ABB RAPID module: P700.mod

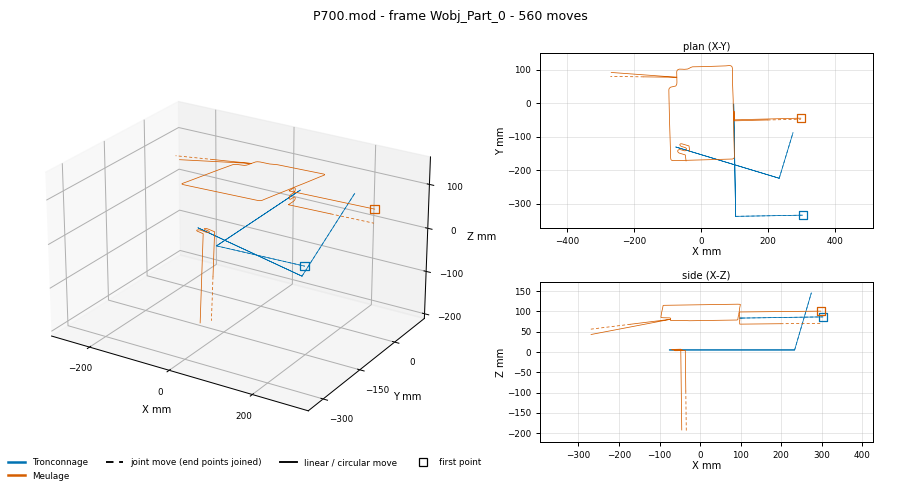
[picture p0: tool path of P700.mod in frame Wobj_Part_0, 560 of 580 moves have a stored position in this frame; points joined in program order, loops and branches not executed]
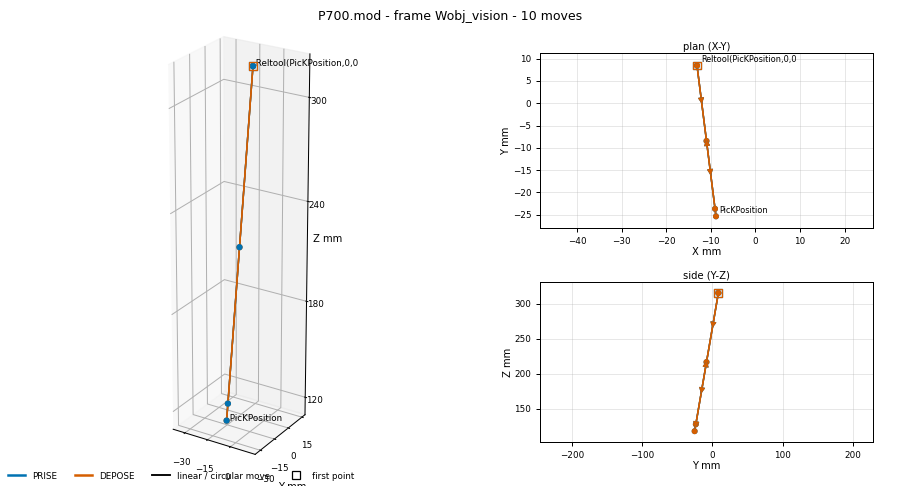
[picture p1: tool path of P700.mod in frame Wobj_vision, 10 of 580 moves have a stored position in this frame; points joined in program order, loops and branches not executed]
MODULE P700

    ! Nom         :P700
    ! Description :
    ! Créé le     :25/05/2023 15:43:03

    LOCAL CONST SPEEDDATA VitesseLente :=[10,500,0,0];
	LOCAL CONST SPEEDDATA VitesseRapide :=[30,500,0,0];
    !
    !Point de prise
    LOCAL PERS Robtarget PicKPosition := [[-8.82508252387174,-25.3604608008818,118.073527161625],[0.0672015502664613,0.699628699637396,0.709367418327075,-0.0529291989496386],[0,0,0,0],[8.999999E+09,8.999999E+09,8.999999E+09,8.999999E+09,8.999999E+09,8.999999E+09]];
	LOCAL PERS Pose Ref := [[0,0,0],[1,0,0,0]];
    !
    !Declaration des points de meulage

    !Tr_meulage_motif_1 : Meulage d'un motif
    LOCAL CONST Robtarget Tr_meulage_motif_1_0 := [[97.6019453125,-49.17523046875,98.798203125],[0.491182031399638,-0.496295254779522,-0.508791654884103,0.50354968377882],[0,0,0,0],[8.999999E+09,8.999999E+09,8.999999E+09,8.999999E+09,8.999999E+09,8.999999E+09]];
    LOCAL CONST Robtarget Tr_meulage_motif_1_1 := [[97.584328125,-48.1753828125,98.7986484375],[0.491182031399638,-0.496295254779522,-0.508791654884103,0.50354968377882],[0,0,0,0],[8.999999E+09,8.999999E+09,8.999999E+09,8.999999E+09,8.999999E+09,8.999999E+09]];
    LOCAL CONST Robtarget Tr_meulage_motif_1_2 := [[97.56671875,-47.1755390625,98.7991015625],[0.491182031399638,-0.496295254779522,-0.508791654884103,0.50354968377882],[0,0,0,0],[8.999999E+09,8.999999E+09,8.999999E+09,8.999999E+09,8.999999E+09,8.999999E+09]];
    LOCAL CONST Robtarget Tr_meulage_motif_1_3 := [[97.549109375,-46.1756953125,98.7995546875],[0.491182031399638,-0.496295254779522,-0.508791654884103,0.50354968377882],[0,0,0,0],[8.999999E+09,8.999999E+09,8.999999E+09,8.999999E+09,8.999999E+09,8.999999E+09]];
    LOCAL CONST Robtarget Tr_meulage_motif_1_4 := [[97.5314921875,-45.1758515625,98.8],[0.491182031399638,-0.496295254779522,-0.508791654884103,0.50354968377882],[0,0,0,0],[8.999999E+09,8.999999E+09,8.999999E+09,8.999999E+09,8.999999E+09,8.999999E+09]];
    LOCAL CONST Robtarget Tr_meulage_motif_1_5 := [[97.5138828125,-44.17600390625,98.800453125],[0.491182031399638,-0.496295254779522,-0.508791654884103,0.50354968377882],[0,0,0,0],[8.999999E+09,8.999999E+09,8.999999E+09,8.999999E+09,8.999999E+09,8.999999E+09]];
    LOCAL CONST Robtarget Tr_meulage_motif_1_6 := [[97.4962734375,-43.17616015625,98.80090625],[0.491182031399638,-0.496295254779522,-0.508791654884103,0.50354968377882],[0,0,0,0],[8.999999E+09,8.999999E+09,8.999999E+09,8.999999E+09,8.999999E+09,8.999999E+09]];
    LOCAL CONST Robtarget Tr_meulage_motif_1_7 := [[97.47865625,-42.17631640625,98.801359375],[0.491182031399638,-0.496295254779522,-0.508791654884103,0.50354968377882],[0,0,0,0],[8.999999E+09,8.999999E+09,8.999999E+09,8.999999E+09,8.999999E+09,8.999999E+09]];
    LOCAL CONST Robtarget Tr_meulage_motif_1_8 := [[97.461046875,-41.17647265625,98.8018046875],[0.491182031399638,-0.496295254779522,-0.508791654884103,0.50354968377882],[0,0,0,0],[8.999999E+09,8.999999E+09,8.999999E+09,8.999999E+09,8.999999E+09,8.999999E+09]];
    LOCAL CONST Robtarget Tr_meulage_motif_1_9 := [[97.4434296875,-40.176625,98.8022578125],[0.491182031399638,-0.496295254779522,-0.508791654884103,0.50354968377882],[0,0,0,0],[8.999999E+09,8.999999E+09,8.999999E+09,8.999999E+09,8.999999E+09,8.999999E+09]];
    LOCAL CONST Robtarget Tr_meulage_motif_1_10 := [[97.4258203125,-39.17678125,98.8027109375],[0.491182031399638,-0.496295254779522,-0.508791654884103,0.50354968377882],[0,0,0,0],[8.999999E+09,8.999999E+09,8.999999E+09,8.999999E+09,8.999999E+09,8.999999E+09]];
    LOCAL CONST Robtarget Tr_meulage_motif_1_11 := [[97.4082109375,-38.1769375,98.80315625],[0.491182031399638,-0.496295254779522,-0.508791654884103,0.50354968377882],[0,0,0,0],[8.999999E+09,8.999999E+09,8.999999E+09,8.999999E+09,8.999999E+09,8.999999E+09]];
    LOCAL CONST Robtarget Tr_meulage_motif_1_12 := [[97.39059375,-37.17709375,98.803609375],[0.491182031399638,-0.496295254779522,-0.508791654884103,0.50354968377882],[0,0,0,0],[8.999999E+09,8.999999E+09,8.999999E+09,8.999999E+09,8.999999E+09,8.999999E+09]];
    LOCAL CONST Robtarget Tr_meulage_motif_1_13 := [[97.372984375,-36.17724609375,98.8040625],[0.491182031399638,-0.496295254779522,-0.508791654884103,0.50354968377882],[0,0,0,0],[8.999999E+09,8.999999E+09,8.999999E+09,8.999999E+09,8.999999E+09,8.999999E+09]];
    LOCAL CONST Robtarget Tr_meulage_motif_1_14 := [[97.3553671875,-35.17740234375,98.8045078125],[0.491182031399638,-0.496295254779522,-0.508791654884103,0.50354968377882],[0,0,0,0],[8.999999E+09,8.999999E+09,8.999999E+09,8.999999E+09,8.999999E+09,8.999999E+09]];
    LOCAL CONST Robtarget Tr_meulage_motif_1_15 := [[97.3377578125,-34.17755859375,98.8049609375],[0.491182031399638,-0.496295254779522,-0.508791654884103,0.50354968377882],[0,0,0,0],[8.999999E+09,8.999999E+09,8.999999E+09,8.999999E+09,8.999999E+09,8.999999E+09]];
    LOCAL CONST Robtarget Tr_meulage_motif_1_16 := [[97.3201484375,-33.1777109375,98.8054140625],[0.491182031399638,-0.496295254779522,-0.508791654884103,0.50354968377882],[0,0,0,0],[8.999999E+09,8.999999E+09,8.999999E+09,8.999999E+09,8.999999E+09,8.999999E+09]];
    LOCAL CONST Robtarget Tr_meulage_motif_1_17 := [[97.30253125,-32.1778671875,98.805859375],[0.491182031399638,-0.496295254779522,-0.508791654884103,0.50354968377882],[0,0,0,0],[8.999999E+09,8.999999E+09,8.999999E+09,8.999999E+09,8.999999E+09,8.999999E+09]];
    LOCAL CONST Robtarget Tr_meulage_motif_1_18 := [[97.284921875,-31.1780234375,98.8063125],[0.491182031399638,-0.496295254779522,-0.508791654884103,0.50354968377882],[0,0,0,0],[8.999999E+09,8.999999E+09,8.999999E+09,8.999999E+09,8.999999E+09,8.999999E+09]];
    LOCAL CONST Robtarget Tr_meulage_motif_1_19 := [[97.2673046875,-30.178177734375,98.806765625],[0.491182031399638,-0.496295254779522,-0.508791654884103,0.50354968377882],[0,0,0,0],[8.999999E+09,8.999999E+09,8.999999E+09,8.999999E+09,8.999999E+09,8.999999E+09]];
    LOCAL CONST Robtarget Tr_meulage_motif_1_20 := [[97.2514296875,-29.18569140625,98.6966328125],[0.491182031399638,-0.496295254779522,-0.508791654884103,0.50354968377882],[0,0,0,0],[8.999999E+09,8.999999E+09,8.999999E+09,8.999999E+09,8.999999E+09,8.999999E+09]];
    LOCAL CONST Robtarget Tr_meulage_motif_1_21 := [[97.237828125,-28.239189453125,98.485890625],[0.491182031399638,-0.496295254779522,-0.508791654884103,0.50354968377882],[0,0,0,0],[8.999999E+09,8.999999E+09,8.999999E+09,8.999999E+09,8.999999E+09,8.999999E+09]];
    LOCAL CONST Robtarget Tr_meulage_motif_1_22 := [[97.2267578125,-27.38641015625,98.2144609375],[0.491182031399638,-0.496295254779522,-0.508791654884103,0.50354968377882],[0,0,0,0],[8.999999E+09,8.999999E+09,8.999999E+09,8.999999E+09,8.999999E+09,8.999999E+09]];
    LOCAL CONST Robtarget Tr_meulage_motif_1_23 := [[97.2175625,-26.63639453125,97.938890625],[0.491182031399638,-0.496295254779522,-0.508791654884103,0.50354968377882],[0,0,0,0],[8.999999E+09,8.999999E+09,8.999999E+09,8.999999E+09,8.999999E+09,8.999999E+09]];
    LOCAL CONST Robtarget Tr_meulage_motif_1_24 := [[97.2071171875,-25.535068359375,97.323328125],[0.491182031399638,-0.496295254779522,-0.508791654884103,0.50354968377882],[0,0,0,0],[8.999999E+09,8.999999E+09,8.999999E+09,8.999999E+09,8.999999E+09,8.999999E+09]];
    LOCAL CONST Robtarget Tr_meulage_motif_1_25 := [[97.2013984375,-24.51075390625,96.47621875],[0.491182031399638,-0.496295254779522,-0.508791654884103,0.50354968377882],[0,0,0,0],[8.999999E+09,8.999999E+09,8.999999E+09,8.999999E+09,8.999999E+09,8.999999E+09]];
    LOCAL CONST Robtarget Tr_meulage_motif_1_26 := [[97.2013359375,-23.66250390625,95.4528359375],[0.491182031399638,-0.496295254779522,-0.508791654884103,0.50354968377882],[0,0,0,0],[8.999999E+09,8.999999E+09,8.999999E+09,8.999999E+09,8.999999E+09,8.999999E+09]];
    LOCAL CONST Robtarget Tr_meulage_motif_1_27 := [[97.208953125,-23.173634765625,94.336984375],[0.491182031399638,-0.496295254779522,-0.508791654884103,0.50354968377882],[0,0,0,0],[8.999999E+09,8.999999E+09,8.999999E+09,8.999999E+09,8.999999E+09,8.999999E+09]];
    LOCAL CONST Robtarget Tr_meulage_motif_1_28 := [[97.2185859375,-23.1460859375,93.6411015625],[0.491182031399638,-0.496295254779522,-0.508791654884103,0.50354968377882],[0,0,0,0],[8.999999E+09,8.999999E+09,8.999999E+09,8.999999E+09,8.999999E+09,8.999999E+09]];
    LOCAL CONST Robtarget Tr_meulage_motif_1_29 := [[97.2281875,-23.145619140625,92.979921875],[0.491182031399638,-0.496295254779522,-0.508791654884103,0.50354968377882],[0,0,0,0],[8.999999E+09,8.999999E+09,8.999999E+09,8.999999E+09,8.999999E+09,8.999999E+09]];
    LOCAL CONST Robtarget Tr_meulage_motif_1_30 := [[97.2387578125,-23.200017578125,92.318875],[0.491182031399638,-0.496295254779522,-0.508791654884103,0.50354968377882],[0,0,0,0],[8.999999E+09,8.999999E+09,8.999999E+09,8.999999E+09,8.999999E+09,8.999999E+09]];
    LOCAL CONST Robtarget Tr_meulage_motif_1_31 := [[97.2635390625,-23.697380859375,91.217015625],[0.491182031399638,-0.496295254779522,-0.508791654884103,0.50354968377882],[0,0,0,0],[8.999999E+09,8.999999E+09,8.999999E+09,8.999999E+09,8.999999E+09,8.999999E+09]];
    LOCAL CONST Robtarget Tr_meulage_motif_1_32 := [[97.2932421875,-24.553162109375,90.210109375],[0.491182031399638,-0.496295254779522,-0.508791654884103,0.50354968377882],[0,0,0,0],[8.999999E+09,8.999999E+09,8.999999E+09,8.999999E+09,8.999999E+09,8.999999E+09]];
    LOCAL CONST Robtarget Tr_meulage_motif_1_33 := [[97.3233125,-25.57582421875,89.3808671875],[0.491182031399638,-0.496295254779522,-0.508791654884103,0.50354968377882],[0,0,0,0],[8.999999E+09,8.999999E+09,8.999999E+09,8.999999E+09,8.999999E+09,8.999999E+09]];
    LOCAL CONST Robtarget Tr_meulage_motif_1_34 := [[97.34115625,-26.26253125,88.98484375],[0.491182031399638,-0.496295254779522,-0.508791654884103,0.50354968377882],[0,0,0,0],[8.999999E+09,8.999999E+09,8.999999E+09,8.999999E+09,8.999999E+09,8.999999E+09]];
    LOCAL CONST Robtarget Tr_meulage_motif_1_35 := [[97.368640625,-27.420162109375,88.49684375],[0.491182031399638,-0.496295254779522,-0.508791654884103,0.50354968377882],[0,0,0,0],[8.999999E+09,8.999999E+09,8.999999E+09,8.999999E+09,8.999999E+09,8.999999E+09]];
    LOCAL CONST Robtarget Tr_meulage_motif_1_36 := [[97.387359375,-28.264876953125,88.2323984375],[0.491182031399638,-0.496295254779522,-0.508791654884103,0.50354968377882],[0,0,0,0],[8.999999E+09,8.999999E+09,8.999999E+09,8.999999E+09,8.999999E+09,8.999999E+09]];
    LOCAL CONST Robtarget Tr_meulage_motif_1_37 := [[97.4067421875,-29.196587890625,88.02753125],[0.491182031399638,-0.496295254779522,-0.508791654884103,0.50354968377882],[0,0,0,0],[8.999999E+09,8.999999E+09,8.999999E+09,8.999999E+09,8.999999E+09,8.999999E+09]];
    LOCAL CONST Robtarget Tr_meulage_motif_1_38 := [[97.425609375,-30.177919921875,87.9185078125],[0.491182031399638,-0.496295254779522,-0.508791654884103,0.50354968377882],[0,0,0,0],[8.999999E+09,8.999999E+09,8.999999E+09,8.999999E+09,8.999999E+09,8.999999E+09]];
    LOCAL CONST Robtarget Tr_meulage_motif_1_39 := [[97.4446953125,-31.17025,87.8074765625],[0.491182031399638,-0.496295254779522,-0.508791654884103,0.50354968377882],[0,0,0,0],[8.999999E+09,8.999999E+09,8.999999E+09,8.999999E+09,8.999999E+09,8.999999E+09]];
    LOCAL CONST Robtarget Tr_meulage_motif_1_40 := [[97.4623046875,-32.170095703125,87.8070234375],[0.491182031399638,-0.496295254779522,-0.508791654884103,0.50354968377882],[0,0,0,0],[8.999999E+09,8.999999E+09,8.999999E+09,8.999999E+09,8.999999E+09,8.999999E+09]];
    LOCAL CONST Robtarget Tr_meulage_motif_1_41 := [[97.479921875,-33.16994140625,87.806578125],[0.491182031399638,-0.496295254779522,-0.508791654884103,0.50354968377882],[0,0,0,0],[8.999999E+09,8.999999E+09,8.999999E+09,8.999999E+09,8.999999E+09,8.999999E+09]];
    LOCAL CONST Robtarget Tr_meulage_motif_1_42 := [[97.49753125,-34.16978515625,87.806125],[0.491182031399638,-0.496295254779522,-0.508791654884103,0.50354968377882],[0,0,0,0],[8.999999E+09,8.999999E+09,8.999999E+09,8.999999E+09,8.999999E+09,8.999999E+09]];
    LOCAL CONST Robtarget Tr_meulage_motif_1_43 := [[97.515140625,-35.16962890625,87.805671875],[0.491182031399638,-0.496295254779522,-0.508791654884103,0.50354968377882],[0,0,0,0],[8.999999E+09,8.999999E+09,8.999999E+09,8.999999E+09,8.999999E+09,8.999999E+09]];
    LOCAL CONST Robtarget Tr_meulage_motif_1_44 := [[97.5327578125,-36.1694765625,87.8052265625],[0.491182031399638,-0.496295254779522,-0.508791654884103,0.50354968377882],[0,0,0,0],[8.999999E+09,8.999999E+09,8.999999E+09,8.999999E+09,8.999999E+09,8.999999E+09]];
    LOCAL CONST Robtarget Tr_meulage_motif_1_45 := [[97.5503671875,-37.1693203125,87.8047734375],[0.491182031399638,-0.496295254779522,-0.508791654884103,0.50354968377882],[0,0,0,0],[8.999999E+09,8.999999E+09,8.999999E+09,8.999999E+09,8.999999E+09,8.999999E+09]];
    LOCAL CONST Robtarget Tr_meulage_motif_1_46 := [[97.567984375,-38.1691640625,87.8043203125],[0.491182031399638,-0.496295254779522,-0.508791654884103,0.50354968377882],[0,0,0,0],[8.999999E+09,8.999999E+09,8.999999E+09,8.999999E+09,8.999999E+09,8.999999E+09]];
    LOCAL CONST Robtarget Tr_meulage_motif_1_47 := [[97.58559375,-39.1690078125,87.8038671875],[0.491182031399638,-0.496295254779522,-0.508791654884103,0.50354968377882],[0,0,0,0],[8.999999E+09,8.999999E+09,8.999999E+09,8.999999E+09,8.999999E+09,8.999999E+09]];
    LOCAL CONST Robtarget Tr_meulage_motif_1_48 := [[97.603203125,-40.16885546875,87.803421875],[0.491182031399638,-0.496295254779522,-0.508791654884103,0.50354968377882],[0,0,0,0],[8.999999E+09,8.999999E+09,8.999999E+09,8.999999E+09,8.999999E+09,8.999999E+09]];
    LOCAL CONST Robtarget Tr_meulage_motif_1_49 := [[97.6208203125,-41.16869921875,87.80296875],[0.491182031399638,-0.496295254779522,-0.508791654884103,0.50354968377882],[0,0,0,0],[8.999999E+09,8.999999E+09,8.999999E+09,8.999999E+09,8.999999E+09,8.999999E+09]];
    LOCAL CONST Robtarget Tr_meulage_motif_1_50 := [[97.6384296875,-42.16854296875,87.802515625],[0.491182031399638,-0.496295254779522,-0.508791654884103,0.50354968377882],[0,0,0,0],[8.999999E+09,8.999999E+09,8.999999E+09,8.999999E+09,8.999999E+09,8.999999E+09]];
    LOCAL CONST Robtarget Tr_meulage_motif_1_51 := [[97.657515625,-43.160875,87.6914921875],[0.491182031399638,-0.496295254779522,-0.508791654884103,0.50354968377882],[0,0,0,0],[8.999999E+09,8.999999E+09,8.999999E+09,8.999999E+09,8.999999E+09,8.999999E+09]];
    LOCAL CONST Robtarget Tr_meulage_motif_1_52 := [[97.6772578125,-44.107078125,87.4798984375],[0.491182031399638,-0.496295254779522,-0.508791654884103,0.50354968377882],[0,0,0,0],[8.999999E+09,8.999999E+09,8.999999E+09,8.999999E+09,8.999999E+09,8.999999E+09]];
    LOCAL CONST Robtarget Tr_meulage_motif_1_53 := [[97.6962265625,-44.95947265625,87.2076953125],[0.491182031399638,-0.496295254779522,-0.508791654884103,0.50354968377882],[0,0,0,0],[8.999999E+09,8.999999E+09,8.999999E+09,8.999999E+09,8.999999E+09,8.999999E+09]];
    LOCAL CONST Robtarget Tr_meulage_motif_1_54 := [[97.713171875,-45.6706484375,86.90325],[0.491182031399638,-0.496295254779522,-0.508791654884103,0.50354968377882],[0,0,0,0],[8.999999E+09,8.999999E+09,8.999999E+09,8.999999E+09,8.999999E+09,8.999999E+09]];
    LOCAL CONST Robtarget Tr_meulage_motif_1_55 := [[97.741015625,-46.70448828125,86.240328125],[0.491182031399638,-0.496295254779522,-0.508791654884103,0.50354968377882],[0,0,0,0],[8.999999E+09,8.999999E+09,8.999999E+09,8.999999E+09,8.999999E+09,8.999999E+09]];
    LOCAL CONST Robtarget Tr_meulage_motif_1_56 := [[97.77,-47.6056484375,85.338078125],[0.491182031399638,-0.496295254779522,-0.508791654884103,0.50354968377882],[0,0,0,0],[8.999999E+09,8.999999E+09,8.999999E+09,8.999999E+09,8.999999E+09,8.999999E+09]];
    LOCAL CONST Robtarget Tr_meulage_motif_1_57 := [[97.7946171875,-48.13979296875,84.2919140625],[0.491182031399638,-0.496295254779522,-0.508791654884103,0.50354968377882],[0,0,0,0],[8.999999E+09,8.999999E+09,8.999999E+09,8.999999E+09,8.999999E+09,8.999999E+09]];
    LOCAL CONST Robtarget Tr_meulage_motif_1_58 := [[97.8079375,-48.3240546875,83.5986875],[0.491182031399638,-0.496295254779522,-0.508791654884103,0.50354968377882],[0,0,0,0],[8.999999E+09,8.999999E+09,8.999999E+09,8.999999E+09,8.999999E+09,8.999999E+09]];
    LOCAL CONST Robtarget Tr_meulage_motif_1_59 := [[97.82025,-48.38734765625,82.8287421875],[0.491182031399638,-0.496295254779522,-0.508791654884103,0.50354968377882],[0,0,0,0],[8.999999E+09,8.999999E+09,8.999999E+09,8.999999E+09,8.999999E+09,8.999999E+09]];
    LOCAL CONST Robtarget Tr_meulage_motif_1_60 := [[97.83025,-48.319875,82.0589765625],[0.491182031399638,-0.496295254779522,-0.508791654884103,0.50354968377882],[0,0,0,0],[8.999999E+09,8.999999E+09,8.999999E+09,8.999999E+09,8.999999E+09,8.999999E+09]];
    LOCAL CONST Robtarget Tr_meulage_motif_1_61 := [[97.8389609375,-47.8995625,80.95103125],[0.491182031399638,-0.496295254779522,-0.508791654884103,0.50354968377882],[0,0,0,0],[8.999999E+09,8.999999E+09,8.999999E+09,8.999999E+09,8.999999E+09,8.999999E+09]];
    LOCAL CONST Robtarget Tr_meulage_motif_1_62 := [[97.840171875,-47.48490234375,80.36559375],[0.491182031399638,-0.496295254779522,-0.508791654884103,0.50354968377882],[0,0,0,0],[8.999999E+09,8.999999E+09,8.999999E+09,8.999999E+09,8.999999E+09,8.999999E+09]];
    LOCAL CONST Robtarget Tr_meulage_motif_1_63 := [[97.8374296875,-46.5972890625,79.4789609375],[0.491182031399638,-0.496295254779522,-0.508791654884103,0.50354968377882],[0,0,0,0],[8.999999E+09,8.999999E+09,8.999999E+09,8.999999E+09,8.999999E+09,8.999999E+09]];
    LOCAL CONST Robtarget Tr_meulage_motif_1_64 := [[97.8331328125,-46.0113984375,79.0649609375],[0.491182031399638,-0.496295254779522,-0.508791654884103,0.50354968377882],[0,0,0,0],[8.999999E+09,8.999999E+09,8.999999E+09,8.999999E+09,8.999999E+09,8.999999E+09]];
    LOCAL CONST Robtarget Tr_meulage_motif_1_65 := [[97.8213515625,-44.89328125,78.521421875],[0.491182031399638,-0.496295254779522,-0.508791654884103,0.50354968377882],[0,0,0,0],[8.999999E+09,8.999999E+09,8.999999E+09,8.999999E+09,8.999999E+09,8.999999E+09]];
    LOCAL CONST Robtarget Tr_meulage_motif_1_66 := [[97.8111015625,-44.06760546875,78.226328125],[0.491182031399638,-0.496295254779522,-0.508791654884103,0.50354968377882],[0,0,0,0],[8.999999E+09,8.999999E+09,8.999999E+09,8.999999E+09,8.999999E+09,8.999999E+09]];
    LOCAL CONST Robtarget Tr_meulage_motif_1_67 := [[97.79765625,-43.13560546875,78.0223046875],[0.491182031399638,-0.496295254779522,-0.508791654884103,0.50354968377882],[0,0,0,0],[8.999999E+09,8.999999E+09,8.999999E+09,8.999999E+09,8.999999E+09,8.999999E+09]];
    LOCAL CONST Robtarget Tr_meulage_motif_1_68 := [[97.7819453125,-42.15412109375,77.9141640625],[0.491182031399638,-0.496295254779522,-0.508791654884103,0.50354968377882],[0,0,0,0],[8.999999E+09,8.999999E+09,8.999999E+09,8.999999E+09,8.999999E+09,8.999999E+09]];
    LOCAL CONST Robtarget Tr_meulage_motif_1_69 := [[97.7660703125,-41.1616328125,77.8040234375],[0.491182031399638,-0.496295254779522,-0.508791654884103,0.50354968377882],[0,0,0,0],[8.999999E+09,8.999999E+09,8.999999E+09,8.999999E+09,8.999999E+09,8.999999E+09]];
    LOCAL CONST Robtarget Tr_meulage_motif_1_70 := [[97.748453125,-40.1617890625,77.8044765625],[0.491182031399638,-0.496295254779522,-0.508791654884103,0.50354968377882],[0,0,0,0],[8.999999E+09,8.999999E+09,8.999999E+09,8.999999E+09,8.999999E+09,8.999999E+09]];
    LOCAL CONST Robtarget Tr_meulage_motif_1_71 := [[97.73084375,-39.1619453125,77.8049296875],[0.491182031399638,-0.496295254779522,-0.508791654884103,0.50354968377882],[0,0,0,0],[8.999999E+09,8.999999E+09,8.999999E+09,8.999999E+09,8.999999E+09,8.999999E+09]];
    LOCAL CONST Robtarget Tr_meulage_motif_1_72 := [[97.713234375,-38.16209765625,77.8053828125],[0.491182031399638,-0.496295254779522,-0.508791654884103,0.50354968377882],[0,0,0,0],[8.999999E+09,8.999999E+09,8.999999E+09,8.999999E+09,8.999999E+09,8.999999E+09]];
    LOCAL CONST Robtarget Tr_meulage_motif_1_73 := [[97.6956171875,-37.16225390625,77.805828125],[0.491182031399638,-0.496295254779522,-0.508791654884103,0.50354968377882],[0,0,0,0],[8.999999E+09,8.999999E+09,8.999999E+09,8.999999E+09,8.999999E+09,8.999999E+09]];
    LOCAL CONST Robtarget Tr_meulage_motif_1_74 := [[97.6780078125,-36.16241015625,77.80628125],[0.491182031399638,-0.496295254779522,-0.508791654884103,0.50354968377882],[0,0,0,0],[8.999999E+09,8.999999E+09,8.999999E+09,8.999999E+09,8.999999E+09,8.999999E+09]];
    LOCAL CONST Robtarget Tr_meulage_motif_1_75 := [[97.660390625,-35.1625625,77.806734375],[0.491182031399638,-0.496295254779522,-0.508791654884103,0.50354968377882],[0,0,0,0],[8.999999E+09,8.999999E+09,8.999999E+09,8.999999E+09,8.999999E+09,8.999999E+09]];
    LOCAL CONST Robtarget Tr_meulage_motif_1_76 := [[97.64278125,-34.16271875,77.8071796875],[0.491182031399638,-0.496295254779522,-0.508791654884103,0.50354968377882],[0,0,0,0],[8.999999E+09,8.999999E+09,8.999999E+09,8.999999E+09,8.999999E+09,8.999999E+09]];
    LOCAL CONST Robtarget Tr_meulage_motif_1_77 := [[97.625171875,-33.162875,77.8076328125],[0.491182031399638,-0.496295254779522,-0.508791654884103,0.50354968377882],[0,0,0,0],[8.999999E+09,8.999999E+09,8.999999E+09,8.999999E+09,8.999999E+09,8.999999E+09]];
    LOCAL CONST Robtarget Tr_meulage_motif_1_78 := [[97.6075546875,-32.163029296875,77.8080859375],[0.491182031399638,-0.496295254779522,-0.508791654884103,0.50354968377882],[0,0,0,0],[8.999999E+09,8.999999E+09,8.999999E+09,8.999999E+09,8.999999E+09,8.999999E+09]];
    LOCAL CONST Robtarget Tr_meulage_motif_1_79 := [[97.5899453125,-31.163185546875,77.80853125],[0.491182031399638,-0.496295254779522,-0.508791654884103,0.50354968377882],[0,0,0,0],[8.999999E+09,8.999999E+09,8.999999E+09,8.999999E+09,8.999999E+09,8.999999E+09]];
    LOCAL CONST Robtarget Tr_meulage_motif_1_80 := [[97.572328125,-30.16333984375,77.808984375],[0.491182031399638,-0.496295254779522,-0.508791654884103,0.50354968377882],[0,0,0,0],[8.999999E+09,8.999999E+09,8.999999E+09,8.999999E+09,8.999999E+09,8.999999E+09]];
    LOCAL CONST Robtarget Tr_meulage_motif_1_81 := [[97.556453125,-29.170853515625,77.6988515625],[0.491182031399638,-0.496295254779522,-0.508791654884103,0.50354968377882],[0,0,0,0],[8.999999E+09,8.999999E+09,8.999999E+09,8.999999E+09,8.999999E+09,8.999999E+09]];
    LOCAL CONST Robtarget Tr_meulage_motif_1_82 := [[97.5428515625,-28.2243515625,77.488109375],[0.491182031399638,-0.496295254779522,-0.508791654884103,0.50354968377882],[0,0,0,0],[8.999999E+09,8.999999E+09,8.999999E+09,8.999999E+09,8.999999E+09,8.999999E+09]];
    LOCAL CONST Robtarget Tr_meulage_motif_1_83 := [[97.53178125,-27.371572265625,77.2166796875],[0.491182031399638,-0.496295254779522,-0.508791654884103,0.50354968377882],[0,0,0,0],[8.999999E+09,8.999999E+09,8.999999E+09,8.999999E+09,8.999999E+09,8.999999E+09]];
    LOCAL CONST Robtarget Tr_meulage_motif_1_84 := [[97.5225859375,-26.621556640625,76.941109375],[0.491182031399638,-0.496295254779522,-0.508791654884103,0.50354968377882],[0,0,0,0],[8.999999E+09,8.999999E+09,8.999999E+09,8.999999E+09,8.999999E+09,8.999999E+09]];
    LOCAL CONST Robtarget Tr_meulage_motif_1_85 := [[97.512140625,-25.52023046875,76.325546875],[0.491182031399638,-0.496295254779522,-0.508791654884103,0.50354968377882],[0,0,0,0],[8.999999E+09,8.999999E+09,8.999999E+09,8.999999E+09,8.999999E+09,8.999999E+09]];
    LOCAL CONST Robtarget Tr_meulage_motif_1_86 := [[97.506421875,-24.4959140625,75.4784375],[0.491182031399638,-0.496295254779522,-0.508791654884103,0.50354968377882],[0,0,0,0],[8.999999E+09,8.999999E+09,8.999999E+09,8.999999E+09,8.999999E+09,8.999999E+09]];
    LOCAL CONST Robtarget Tr_meulage_motif_1_87 := [[97.5086328125,-23.742841796875,74.413953125],[0.491182031399638,-0.496295254779522,-0.508791654884103,0.50354968377882],[0,0,0,0],[8.999999E+09,8.999999E+09,8.999999E+09,8.999999E+09,8.999999E+09,8.999999E+09]];
    LOCAL CONST Robtarget Tr_meulage_motif_1_88 := [[97.5176328125,-23.336869140625,73.3031953125],[0.491182031399638,-0.496295254779522,-0.508791654884103,0.50354968377882],[0,0,0,0],[8.999999E+09,8.999999E+09,8.999999E+09,8.999999E+09,8.999999E+09,8.999999E+09]];
    LOCAL CONST Robtarget Tr_meulage_motif_1_89 := [[97.5284296875,-23.47397265625,72.7267265625],[0.491182031399638,-0.496295254779522,-0.508791654884103,0.50354968377882],[0,0,0,0],[8.999999E+09,8.999999E+09,8.999999E+09,8.999999E+09,8.999999E+09,8.999999E+09]];
    LOCAL CONST Robtarget Tr_meulage_motif_1_90 := [[97.53415625,-23.53814453125,72.4108828125],[0.491182031399638,-0.496295254779522,-0.508791654884103,0.50354968377882],[0,0,0,0],[8.999999E+09,8.999999E+09,8.999999E+09,8.999999E+09,8.999999E+09,8.999999E+09]];
    LOCAL CONST Robtarget Tr_meulage_motif_1_91 := [[97.5540390625,-23.916974609375,71.50184375],[0.491182031399638,-0.496295254779522,-0.508791654884103,0.50354968377882],[0,0,0,0],[8.999999E+09,8.999999E+09,8.999999E+09,8.999999E+09,8.999999E+09,8.999999E+09]];
    LOCAL CONST Robtarget Tr_meulage_motif_1_92 := [[97.5680859375,-24.276701171875,70.971546875],[0.491182031399638,-0.496295254779522,-0.508791654884103,0.50354968377882],[0,0,0,0],[8.999999E+09,8.999999E+09,8.999999E+09,8.999999E+09,8.999999E+09,8.999999E+09]];
    LOCAL CONST Robtarget Tr_meulage_motif_1_93 := [[97.59846875,-25.368177734375,70.2037890625],[0.491182031399638,-0.496295254779522,-0.508791654884103,0.50354968377882],[0,0,0,0],[8.999999E+09,8.999999E+09,8.999999E+09,8.999999E+09,8.999999E+09,8.999999E+09]];
    LOCAL CONST Robtarget Tr_meulage_motif_1_94 := [[97.618078125,-26.15830859375,69.8116328125],[0.491182031399638,-0.496295254779522,-0.508791654884103,0.50354968377882],[0,0,0,0],[8.999999E+09,8.999999E+09,8.999999E+09,8.999999E+09,8.999999E+09,8.999999E+09]];
    LOCAL CONST Robtarget Tr_meulage_motif_1_95 := [[97.64440625,-27.335478515625,69.426546875],[0.491182031399638,-0.496295254779522,-0.508791654884103,0.50354968377882],[0,0,0,0],[8.999999E+09,8.999999E+09,8.999999E+09,8.999999E+09,8.999999E+09,8.999999E+09]];
    LOCAL CONST Robtarget Tr_meulage_motif_1_96 := [[97.663328125,-28.251451171875,69.23440625],[0.491182031399638,-0.496295254779522,-0.508791654884103,0.50354968377882],[0,0,0,0],[8.999999E+09,8.999999E+09,8.999999E+09,8.999999E+09,8.999999E+09,8.999999E+09]];
    LOCAL CONST Robtarget Tr_meulage_motif_1_97 := [[97.68271875,-29.183162109375,69.0295390625],[0.491182031399638,-0.496295254779522,-0.508791654884103,0.50354968377882],[0,0,0,0],[8.999999E+09,8.999999E+09,8.999999E+09,8.999999E+09,8.999999E+09,8.999999E+09]];
    LOCAL CONST Robtarget Tr_meulage_motif_1_98 := [[97.701578125,-30.16449609375,68.920515625],[0.491182031399638,-0.496295254779522,-0.508791654884103,0.50354968377882],[0,0,0,0],[8.999999E+09,8.999999E+09,8.999999E+09,8.999999E+09,8.999999E+09,8.999999E+09]];
    LOCAL CONST Robtarget Tr_meulage_motif_1_99 := [[97.720671875,-31.156826171875,68.809484375],[0.491182031399638,-0.496295254779522,-0.508791654884103,0.50354968377882],[0,0,0,0],[8.999999E+09,8.999999E+09,8.999999E+09,8.999999E+09,8.999999E+09,8.999999E+09]];
    LOCAL CONST Robtarget Tr_meulage_motif_1_100 := [[97.73828125,-32.156669921875,68.80903125],[0.491182031399638,-0.496295254779522,-0.508791654884103,0.50354968377882],[0,0,0,0],[8.999999E+09,8.999999E+09,8.999999E+09,8.999999E+09,8.999999E+09,8.999999E+09]];
    LOCAL CONST Robtarget Tr_meulage_motif_1_101 := [[97.755890625,-33.156515625,68.8085859375],[0.491182031399638,-0.496295254779522,-0.508791654884103,0.50354968377882],[0,0,0,0],[8.999999E+09,8.999999E+09,8.999999E+09,8.999999E+09,8.999999E+09,8.999999E+09]];
    LOCAL CONST Robtarget Tr_meulage_motif_1_102 := [[97.7735078125,-34.156359375,68.8081328125],[0.491182031399638,-0.496295254779522,-0.508791654884103,0.50354968377882],[0,0,0,0],[8.999999E+09,8.999999E+09,8.999999E+09,8.999999E+09,8.999999E+09,8.999999E+09]];
    LOCAL CONST Robtarget Tr_meulage_motif_1_103 := [[97.7911171875,-35.15620703125,68.8076796875],[0.491182031399638,-0.496295254779522,-0.508791654884103,0.50354968377882],[0,0,0,0],[8.999999E+09,8.999999E+09,8.999999E+09,8.999999E+09,8.999999E+09,8.999999E+09]];
    LOCAL CONST Robtarget Tr_meulage_motif_1_104 := [[97.808734375,-36.15605078125,68.807234375],[0.491182031399638,-0.496295254779522,-0.508791654884103,0.50354968377882],[0,0,0,0],[8.999999E+09,8.999999E+09,8.999999E+09,8.999999E+09,8.999999E+09,8.999999E+09]];
    LOCAL CONST Robtarget Tr_meulage_motif_1_105 := [[97.82634375,-37.15589453125,68.80678125],[0.491182031399638,-0.496295254779522,-0.508791654884103,0.50354968377882],[0,0,0,0],[8.999999E+09,8.999999E+09,8.999999E+09,8.999999E+09,8.999999E+09,8.999999E+09]];
    LOCAL CONST Robtarget Tr_meulage_motif_1_106 := [[97.843953125,-38.15573828125,68.806328125],[0.491182031399638,-0.496295254779522,-0.508791654884103,0.50354968377882],[0,0,0,0],[8.999999E+09,8.999999E+09,8.999999E+09,8.999999E+09,8.999999E+09,8.999999E+09]];
    LOCAL CONST Robtarget Tr_meulage_motif_1_107 := [[97.8615703125,-39.1555859375,68.8058828125],[0.491182031399638,-0.496295254779522,-0.508791654884103,0.50354968377882],[0,0,0,0],[8.999999E+09,8.999999E+09,8.999999E+09,8.999999E+09,8.999999E+09,8.999999E+09]];
    LOCAL CONST Robtarget Tr_meulage_motif_1_108 := [[97.8791796875,-40.1554296875,68.8054296875],[0.491182031399638,-0.496295254779522,-0.508791654884103,0.50354968377882],[0,0,0,0],[8.999999E+09,8.999999E+09,8.999999E+09,8.999999E+09,8.999999E+09,8.999999E+09]];
    LOCAL CONST Robtarget Tr_meulage_motif_1_109 := [[97.896796875,-41.1552734375,68.8049765625],[0.491182031399638,-0.496295254779522,-0.508791654884103,0.50354968377882],[0,0,0,0],[8.999999E+09,8.999999E+09,8.999999E+09,8.999999E+09,8.999999E+09,8.999999E+09]];
    LOCAL CONST Robtarget Tr_meulage_motif_1_110 := [[97.91440625,-42.1551171875,68.80453125],[0.491182031399638,-0.496295254779522,-0.508791654884103,0.50354968377882],[0,0,0,0],[8.999999E+09,8.999999E+09,8.999999E+09,8.999999E+09,8.999999E+09,8.999999E+09]];
    LOCAL CONST Robtarget Tr_meulage_motif_1_111 := [[97.932015625,-43.15496484375,68.804078125],[0.491182031399638,-0.496295254779522,-0.508791654884103,0.50354968377882],[0,0,0,0],[8.999999E+09,8.999999E+09,8.999999E+09,8.999999E+09,8.999999E+09,8.999999E+09]];
    LOCAL CONST Robtarget Tr_meulage_motif_1_112 := [[97.9496328125,-44.15480859375,68.803625],[0.491182031399638,-0.496295254779522,-0.508791654884103,0.50354968377882],[0,0,0,0],[8.999999E+09,8.999999E+09,8.999999E+09,8.999999E+09,8.999999E+09,8.999999E+09]];
    LOCAL CONST Robtarget Tr_meulage_motif_1_113 := [[97.9672421875,-45.15465234375,68.8031796875],[0.491182031399638,-0.496295254779522,-0.508791654884103,0.50354968377882],[0,0,0,0],[8.999999E+09,8.999999E+09,8.999999E+09,8.999999E+09,8.999999E+09,8.999999E+09]];
    LOCAL CONST Robtarget Tr_meulage_motif_1_114 := [[97.984859375,-46.15449609375,68.8027265625],[0.491182031399638,-0.496295254779522,-0.508791654884103,0.50354968377882],[0,0,0,0],[8.999999E+09,8.999999E+09,8.999999E+09,8.999999E+09,8.999999E+09,8.999999E+09]];
    LOCAL CONST Robtarget Tr_meulage_motif_1_115 := [[98.00246875,-47.15434375,68.8022734375],[0.491182031399638,-0.496295254779522,-0.508791654884103,0.50354968377882],[0,0,0,0],[8.999999E+09,8.999999E+09,8.999999E+09,8.999999E+09,8.999999E+09,8.999999E+09]];
    LOCAL CONST Robtarget Tr_meulage_motif_1_116 := [[98.020078125,-48.1541875,68.8018203125],[0.491182031399638,-0.496295254779522,-0.508791654884103,0.50354968377882],[0,0,0,0],[8.999999E+09,8.999999E+09,8.999999E+09,8.999999E+09,8.999999E+09,8.999999E+09]];
    LOCAL CONST Robtarget Tr_meulage_motif_1_117 := [[98.0376953125,-49.15403125,68.801375],[0.491182031399638,-0.496295254779522,-0.508791654884103,0.50354968377882],[0,0,0,0],[8.999999E+09,8.999999E+09,8.999999E+09,8.999999E+09,8.999999E+09,8.999999E+09]];
    LOCAL CONST Robtarget Tr_meulage_motif_1_118 := [[98.0553046875,-50.15387890625,68.800921875],[0.491182031399638,-0.496295254779522,-0.508791654884103,0.50354968377882],[0,0,0,0],[8.999999E+09,8.999999E+09,8.999999E+09,8.999999E+09,8.999999E+09,8.999999E+09]];
    LOCAL CONST Robtarget Tr_meulage_motif_1_119 := [[98.0729140625,-51.15372265625,68.80046875],[0.491182031399638,-0.496295254779522,-0.508791654884103,0.50354968377882],[0,0,0,0],[8.999999E+09,8.999999E+09,8.999999E+09,8.999999E+09,8.999999E+09,8.999999E+09]];
    LOCAL CONST Robtarget Tr_meulage_motif_1_120 := [[98.09053125,-52.15356640625,68.8000234375],[0.491182031399638,-0.496295254779522,-0.508791654884103,0.50354968377882],[0,0,0,0],[8.999999E+09,8.999999E+09,8.999999E+09,8.999999E+09,8.999999E+09,8.999999E+09]];

    !Tr_meulage_motif_2 : Meulage d'un motif
    LOCAL CONST Robtarget Tr_meulage_motif_2_0 := [[-47.74959375,-153.919828125,6.9766171875],[-0.000274293000079729,0.00605508420207388,-0.0452523792521339,-0.998957197727048],[0,0,0,0],[8.999999E+09,8.999999E+09,8.999999E+09,8.999999E+09,8.999999E+09,8.999999E+09]];
    LOCAL CONST Robtarget Tr_meulage_motif_2_1 := [[-48.707671875,-153.634703125,6.94869921875],[-0.000274293000079729,0.00605508420207388,-0.0452523792521339,-0.998957197727048],[0,0,0,0],[8.999999E+09,8.999999E+09,8.999999E+09,8.999999E+09,8.999999E+09,8.999999E+09]];
    LOCAL CONST Robtarget Tr_meulage_motif_2_2 := [[-49.66575390625,-153.3495625,6.92078173828125],[-0.000274293000079729,0.00605508420207388,-0.0452523792521339,-0.998957197727048],[0,0,0,0],[8.999999E+09,8.999999E+09,8.999999E+09,8.999999E+09,8.999999E+09,8.999999E+09]];
    LOCAL CONST Robtarget Tr_meulage_motif_2_3 := [[-50.6238359375,-153.0644375,6.89286376953125],[-0.000274293000079729,0.00605508420207388,-0.0452523792521339,-0.998957197727048],[0,0,0,0],[8.999999E+09,8.999999E+09,8.999999E+09,8.999999E+09,8.999999E+09,8.999999E+09]];
    LOCAL CONST Robtarget Tr_meulage_motif_2_4 := [[-51.58191796875,-152.779296875,6.8649462890625],[-0.000274293000079729,0.00605508420207388,-0.0452523792521339,-0.998957197727048],[0,0,0,0],[8.999999E+09,8.999999E+09,8.999999E+09,8.999999E+09,8.999999E+09,8.999999E+09]];
    LOCAL CONST Robtarget Tr_meulage_motif_2_5 := [[-52.54,-152.494171875,6.8370283203125],[-0.000274293000079729,0.00605508420207388,-0.0452523792521339,-0.998957197727048],[0,0,0,0],[8.999999E+09,8.999999E+09,8.999999E+09,8.999999E+09,8.999999E+09,8.999999E+09]];
    LOCAL CONST Robtarget Tr_meulage_motif_2_6 := [[-53.498078125,-152.20903125,6.8091103515625],[-0.000274293000079729,0.00605508420207388,-0.0452523792521339,-0.998957197727048],[0,0,0,0],[8.999999E+09,8.999999E+09,8.999999E+09,8.999999E+09,8.999999E+09,8.999999E+09]];
    LOCAL CONST Robtarget Tr_meulage_motif_2_7 := [[-54.45616015625,-151.923890625,6.78119287109375],[-0.000274293000079729,0.00605508420207388,-0.0452523792521339,-0.998957197727048],[0,0,0,0],[8.999999E+09,8.999999E+09,8.999999E+09,8.999999E+09,8.999999E+09,8.999999E+09]];
    LOCAL CONST Robtarget Tr_meulage_motif_2_8 := [[-55.4142421875,-151.638765625,6.75327490234375],[-0.000274293000079729,0.00605508420207388,-0.0452523792521339,-0.998957197727048],[0,0,0,0],[8.999999E+09,8.999999E+09,8.999999E+09,8.999999E+09,8.999999E+09,8.999999E+09]];
    LOCAL CONST Robtarget Tr_meulage_motif_2_9 := [[-56.37232421875,-151.353625,6.72535693359375],[-0.000274293000079729,0.00605508420207388,-0.0452523792521339,-0.998957197727048],[0,0,0,0],[8.999999E+09,8.999999E+09,8.999999E+09,8.999999E+09,8.999999E+09,8.999999E+09]];
    LOCAL CONST Robtarget Tr_meulage_motif_2_10 := [[-57.33040625,-151.0685,6.697439453125],[-0.000274293000079729,0.00605508420207388,-0.0452523792521339,-0.998957197727048],[0,0,0,0],[8.999999E+09,8.999999E+09,8.999999E+09,8.999999E+09,8.999999E+09,8.999999E+09]];
    LOCAL CONST Robtarget Tr_meulage_motif_2_11 := [[-58.288484375,-150.783359375,6.669521484375],[-0.000274293000079729,0.00605508420207388,-0.0452523792521339,-0.998957197727048],[0,0,0,0],[8.999999E+09,8.999999E+09,8.999999E+09,8.999999E+09,8.999999E+09,8.999999E+09]];
    LOCAL CONST Robtarget Tr_meulage_motif_2_12 := [[-59.24656640625,-150.498234375,6.64160400390625],[-0.000274293000079729,0.00605508420207388,-0.0452523792521339,-0.998957197727048],[0,0,0,0],[8.999999E+09,8.999999E+09,8.999999E+09,8.999999E+09,8.999999E+09,8.999999E+09]];
    LOCAL CONST Robtarget Tr_meulage_motif_2_13 := [[-60.2046484375,-150.21309375,6.61368603515625],[-0.000274293000079729,0.00605508420207388,-0.0452523792521339,-0.998957197727048],[0,0,0,0],[8.999999E+09,8.999999E+09,8.999999E+09,8.999999E+09,8.999999E+09,8.999999E+09]];
    LOCAL CONST Robtarget Tr_meulage_motif_2_14 := [[-61.16273046875,-149.92796875,6.58576806640625],[-0.000274293000079729,0.00605508420207388,-0.0452523792521339,-0.998957197727048],[0,0,0,0],[8.999999E+09,8.999999E+09,8.999999E+09,8.999999E+09,8.999999E+09,8.999999E+09]];
    LOCAL CONST Robtarget Tr_meulage_motif_2_15 := [[-62.1208125,-149.642828125,6.5578505859375],[-0.000274293000079729,0.00605508420207388,-0.0452523792521339,-0.998957197727048],[0,0,0,0],[8.999999E+09,8.999999E+09,8.999999E+09,8.999999E+09,8.999999E+09,8.999999E+09]];
    LOCAL CONST Robtarget Tr_meulage_motif_2_16 := [[-63.07889453125,-149.357703125,6.5299326171875],[-0.000274293000079729,0.00605508420207388,-0.0452523792521339,-0.998957197727048],[0,0,0,0],[8.999999E+09,8.999999E+09,8.999999E+09,8.999999E+09,8.999999E+09,8.999999E+09]];
    LOCAL CONST Robtarget Tr_meulage_motif_2_17 := [[-64.03697265625,-149.0725625,6.5020146484375],[-0.000274293000079729,0.00605508420207388,-0.0452523792521339,-0.998957197727048],[0,0,0,0],[8.999999E+09,8.999999E+09,8.999999E+09,8.999999E+09,8.999999E+09,8.999999E+09]];
    LOCAL CONST Robtarget Tr_meulage_motif_2_18 := [[-64.9950546875,-148.7874375,6.47409716796875],[-0.000274293000079729,0.00605508420207388,-0.0452523792521339,-0.998957197727048],[0,0,0,0],[8.999999E+09,8.999999E+09,8.999999E+09,8.999999E+09,8.999999E+09,8.999999E+09]];
    LOCAL CONST Robtarget Tr_meulage_motif_2_19 := [[-65.914328125,-148.399125,6.4346064453125],[-0.000274293000079729,0.00605508420207388,-0.0452523792521339,-0.998957197727048],[0,0,0,0],[8.999999E+09,8.999999E+09,8.999999E+09,8.999999E+09,8.999999E+09,8.999999E+09]];
    LOCAL CONST Robtarget Tr_meulage_motif_2_20 := [[-66.76065625,-147.92815625,6.38568701171875],[-0.000274293000079729,0.00605508420207388,-0.0452523792521339,-0.998957197727048],[0,0,0,0],[8.999999E+09,8.999999E+09,8.999999E+09,8.999999E+09,8.999999E+09,8.999999E+09]];
    LOCAL CONST Robtarget Tr_meulage_motif_2_21 := [[-67.49975,-147.4261875,6.33292431640625],[-0.000274293000079729,0.00605508420207388,-0.0452523792521339,-0.998957197727048],[0,0,0,0],[8.999999E+09,8.999999E+09,8.999999E+09,8.999999E+09,8.999999E+09,8.999999E+09]];
    LOCAL CONST Robtarget Tr_meulage_motif_2_22 := [[-68.139203125,-146.949625,6.2825947265625],[-0.000274293000079729,0.00605508420207388,-0.0452523792521339,-0.998957197727048],[0,0,0,0],[8.999999E+09,8.999999E+09,8.999999E+09,8.999999E+09,8.999999E+09,8.999999E+09]];
    LOCAL CONST Robtarget Tr_meulage_motif_2_23 := [[-69.017609375,-146.04903125,6.1862265625],[-0.000274293000079729,0.00605508420207388,-0.0452523792521339,-0.998957197727048],[0,0,0,0],[8.999999E+09,8.999999E+09,8.999999E+09,8.999999E+09,8.999999E+09,8.999999E+09]];
    LOCAL CONST Robtarget Tr_meulage_motif_2_24 := [[-69.755734375,-144.95,6.06735009765625],[-0.000274293000079729,0.00605508420207388,-0.0452523792521339,-0.998957197727048],[0,0,0,0],[8.999999E+09,8.999999E+09,8.999999E+09,8.999999E+09,8.999999E+09,8.999999E+09]];
    LOCAL CONST Robtarget Tr_meulage_motif_2_25 := [[-70.274546875,-143.733421875,5.934623046875],[-0.000274293000079729,0.00605508420207388,-0.0452523792521339,-0.998957197727048],[0,0,0,0],[8.999999E+09,8.999999E+09,8.999999E+09,8.999999E+09,8.999999E+09,8.999999E+09]];
    LOCAL CONST Robtarget Tr_meulage_motif_2_26 := [[-70.422484375,-142.531453125,5.80209912109375],[-0.000274293000079729,0.00605508420207388,-0.0452523792521339,-0.998957197727048],[0,0,0,0],[8.999999E+09,8.999999E+09,8.999999E+09,8.999999E+09,8.999999E+09,8.999999E+09]];
    LOCAL CONST Robtarget Tr_meulage_motif_2_27 := [[-70.2490390625,-141.8610625,5.72720947265625],[-0.000274293000079729,0.00605508420207388,-0.0452523792521339,-0.998957197727048],[0,0,0,0],[8.999999E+09,8.999999E+09,8.999999E+09,8.999999E+09,8.999999E+09,8.999999E+09]];
    LOCAL CONST Robtarget Tr_meulage_motif_2_28 := [[-70.059609375,-141.231453125,5.6567734375],[-0.000274293000079729,0.00605508420207388,-0.0452523792521339,-0.998957197727048],[0,0,0,0],[8.999999E+09,8.999999E+09,8.999999E+09,8.999999E+09,8.999999E+09,8.999999E+09]];
    LOCAL CONST Robtarget Tr_meulage_motif_2_29 := [[-69.8176484375,-140.617640625,5.5878857421875],[-0.000274293000079729,0.00605508420207388,-0.0452523792521339,-0.998957197727048],[0,0,0,0],[8.999999E+09,8.999999E+09,8.999999E+09,8.999999E+09,8.999999E+09,8.999999E+09]];
    LOCAL CONST Robtarget Tr_meulage_motif_2_30 := [[-69.0246953125,-139.710671875,5.4844375],[-0.000274293000079729,0.00605508420207388,-0.0452523792521339,-0.998957197727048],[0,0,0,0],[8.999999E+09,8.999999E+09,8.999999E+09,8.999999E+09,8.999999E+09,8.999999E+09]];
    LOCAL CONST Robtarget Tr_meulage_motif_2_31 := [[-67.915609375,-138.99646875,5.40112744140625],[-0.000274293000079729,0.00605508420207388,-0.0452523792521339,-0.998957197727048],[0,0,0,0],[8.999999E+09,8.999999E+09,8.999999E+09,8.999999E+09,8.999999E+09,8.999999E+09]];
    LOCAL CONST Robtarget Tr_meulage_motif_2_32 := [[-66.69765625,-138.4990625,5.3414072265625],[-0.000274293000079729,0.00605508420207388,-0.0452523792521339,-0.998957197727048],[0,0,0,0],[8.999999E+09,8.999999E+09,8.999999E+09,8.999999E+09,8.999999E+09,8.999999E+09]];
    LOCAL CONST Robtarget Tr_meulage_motif_2_33 := [[-65.9259921875,-138.31815625,5.3184345703125],[-0.000274293000079729,0.00605508420207388,-0.0452523792521339,-0.998957197727048],[0,0,0,0],[8.999999E+09,8.999999E+09,8.999999E+09,8.999999E+09,8.999999E+09,8.999999E+09]];
    LOCAL CONST Robtarget Tr_meulage_motif_2_34 := [[-64.67671875,-138.1841875,5.2988359375],[-0.000274293000079729,0.00605508420207388,-0.0452523792521339,-0.998957197727048],[0,0,0,0],[8.999999E+09,8.999999E+09,8.999999E+09,8.999999E+09,8.999999E+09,8.999999E+09]];
    LOCAL CONST Robtarget Tr_meulage_motif_2_35 := [[-63.79145703125,-138.1736875,5.29429638671875],[-0.000274293000079729,0.00605508420207388,-0.0452523792521339,-0.998957197727048],[0,0,0,0],[8.999999E+09,8.999999E+09,8.999999E+09,8.999999E+09,8.999999E+09,8.999999E+09]];
    LOCAL CONST Robtarget Tr_meulage_motif_2_36 := [[-62.83994921875,-138.244734375,5.29853564453125],[-0.000274293000079729,0.00605508420207388,-0.0452523792521339,-0.998957197727048],[0,0,0,0],[8.999999E+09,8.999999E+09,8.999999E+09,8.999999E+09,8.999999E+09,8.999999E+09]];
    LOCAL CONST Robtarget Tr_meulage_motif_2_37 := [[-61.86842578125,-138.42121875,5.31437158203125],[-0.000274293000079729,0.00605508420207388,-0.0452523792521339,-0.998957197727048],[0,0,0,0],[8.999999E+09,8.999999E+09,8.999999E+09,8.999999E+09,8.999999E+09,8.999999E+09]];
    LOCAL CONST Robtarget Tr_meulage_motif_2_38 := [[-60.8857890625,-138.598921875,5.33030126953125],[-0.000274293000079729,0.00605508420207388,-0.0452523792521339,-0.998957197727048],[0,0,0,0],[8.999999E+09,8.999999E+09,8.999999E+09,8.999999E+09,8.999999E+09,8.999999E+09]];
    LOCAL CONST Robtarget Tr_meulage_motif_2_39 := [[-59.92770703125,-138.8840625,5.35821875],[-0.000274293000079729,0.00605508420207388,-0.0452523792521339,-0.998957197727048],[0,0,0,0],[8.999999E+09,8.999999E+09,8.999999E+09,8.999999E+09,8.999999E+09,8.999999E+09]];
    LOCAL CONST Robtarget Tr_meulage_motif_2_40 := [[-58.969625,-139.1691875,5.38613671875],[-0.000274293000079729,0.00605508420207388,-0.0452523792521339,-0.998957197727048],[0,0,0,0],[8.999999E+09,8.999999E+09,8.999999E+09,8.999999E+09,8.999999E+09,8.999999E+09]];
    LOCAL CONST Robtarget Tr_meulage_motif_2_41 := [[-58.01154296875,-139.454328125,5.4140546875],[-0.000274293000079729,0.00605508420207388,-0.0452523792521339,-0.998957197727048],[0,0,0,0],[8.999999E+09,8.999999E+09,8.999999E+09,8.999999E+09,8.999999E+09,8.999999E+09]];
    LOCAL CONST Robtarget Tr_meulage_motif_2_42 := [[-57.0534609375,-139.73946875,5.44197216796875],[-0.000274293000079729,0.00605508420207388,-0.0452523792521339,-0.998957197727048],[0,0,0,0],[8.999999E+09,8.999999E+09,8.999999E+09,8.999999E+09,8.999999E+09,8.999999E+09]];
    LOCAL CONST Robtarget Tr_meulage_motif_2_43 := [[-56.0953828125,-140.02459375,5.46989013671875],[-0.000274293000079729,0.00605508420207388,-0.0452523792521339,-0.998957197727048],[0,0,0,0],[8.999999E+09,8.999999E+09,8.999999E+09,8.999999E+09,8.999999E+09,8.999999E+09]];
    LOCAL CONST Robtarget Tr_meulage_motif_2_44 := [[-55.13730078125,-140.309734375,5.49780810546875],[-0.000274293000079729,0.00605508420207388,-0.0452523792521339,-0.998957197727048],[0,0,0,0],[8.999999E+09,8.999999E+09,8.999999E+09,8.999999E+09,8.999999E+09,8.999999E+09]];
    LOCAL CONST Robtarget Tr_meulage_motif_2_45 := [[-54.17921875,-140.594859375,5.5257255859375],[-0.000274293000079729,0.00605508420207388,-0.0452523792521339,-0.998957197727048],[0,0,0,0],[8.999999E+09,8.999999E+09,8.999999E+09,8.999999E+09,8.999999E+09,8.999999E+09]];
    LOCAL CONST Robtarget Tr_meulage_motif_2_46 := [[-53.22113671875,-140.88,5.5536435546875],[-0.000274293000079729,0.00605508420207388,-0.0452523792521339,-0.998957197727048],[0,0,0,0],[8.999999E+09,8.999999E+09,8.999999E+09,8.999999E+09,8.999999E+09,8.999999E+09]];
    LOCAL CONST Robtarget Tr_meulage_motif_2_47 := [[-52.2630546875,-141.165125,5.58156103515625],[-0.000274293000079729,0.00605508420207388,-0.0452523792521339,-0.998957197727048],[0,0,0,0],[8.999999E+09,8.999999E+09,8.999999E+09,8.999999E+09,8.999999E+09,8.999999E+09]];
    LOCAL CONST Robtarget Tr_meulage_motif_2_48 := [[-51.3049765625,-141.450265625,5.60947900390625],[-0.000274293000079729,0.00605508420207388,-0.0452523792521339,-0.998957197727048],[0,0,0,0],[8.999999E+09,8.999999E+09,8.999999E+09,8.999999E+09,8.999999E+09,8.999999E+09]];
    LOCAL CONST Robtarget Tr_meulage_motif_2_49 := [[-50.3223359375,-141.62796875,5.62540869140625],[-0.000274293000079729,0.00605508420207388,-0.0452523792521339,-0.998957197727048],[0,0,0,0],[8.999999E+09,8.999999E+09,8.999999E+09,8.999999E+09,8.999999E+09,8.999999E+09]];
    LOCAL CONST Robtarget Tr_meulage_motif_2_50 := [[-49.355015625,-141.696765625,5.62933740234375],[-0.000274293000079729,0.00605508420207388,-0.0452523792521339,-0.998957197727048],[0,0,0,0],[8.999999E+09,8.999999E+09,8.999999E+09,8.999999E+09,8.999999E+09,8.999999E+09]];
    LOCAL CONST Robtarget Tr_meulage_motif_2_51 := [[-48.4601640625,-141.6810625,5.62418701171875],[-0.000274293000079729,0.00605508420207388,-0.0452523792521339,-0.998957197727048],[0,0,0,0],[8.999999E+09,8.999999E+09,8.999999E+09,8.999999E+09,8.999999E+09,8.999999E+09]];
    LOCAL CONST Robtarget Tr_meulage_motif_2_52 := [[-47.691359375,-141.59434375,5.61165185546875],[-0.000274293000079729,0.00605508420207388,-0.0452523792521339,-0.998957197727048],[0,0,0,0],[8.999999E+09,8.999999E+09,8.999999E+09,8.999999E+09,8.999999E+09,8.999999E+09]];
    LOCAL CONST Robtarget Tr_meulage_motif_2_53 := [[-46.51045703125,-141.25846875,5.56995947265625],[-0.000274293000079729,0.00605508420207388,-0.0452523792521339,-0.998957197727048],[0,0,0,0],[8.999999E+09,8.999999E+09,8.999999E+09,8.999999E+09,8.999999E+09,8.999999E+09]];
    LOCAL CONST Robtarget Tr_meulage_motif_2_54 := [[-45.38794921875,-140.656859375,5.4990654296875],[-0.000274293000079729,0.00605508420207388,-0.0452523792521339,-0.998957197727048],[0,0,0,0],[8.999999E+09,8.999999E+09,8.999999E+09,8.999999E+09,8.999999E+09,8.999999E+09]];
    LOCAL CONST Robtarget Tr_meulage_motif_2_55 := [[-44.57574609375,-139.813421875,5.402578125],[-0.000274293000079729,0.00605508420207388,-0.0452523792521339,-0.998957197727048],[0,0,0,0],[8.999999E+09,8.999999E+09,8.999999E+09,8.999999E+09,8.999999E+09,8.999999E+09]];
    LOCAL CONST Robtarget Tr_meulage_motif_2_56 := [[-44.20012109375,-139.2060625,5.3338955078125],[-0.000274293000079729,0.00605508420207388,-0.0452523792521339,-0.998957197727048],[0,0,0,0],[8.999999E+09,8.999999E+09,8.999999E+09,8.999999E+09,8.999999E+09,8.999999E+09]];
    LOCAL CONST Robtarget Tr_meulage_motif_2_57 := [[-43.91837109375,-138.491109375,5.253658203125],[-0.000274293000079729,0.00605508420207388,-0.0452523792521339,-0.998957197727048],[0,0,0,0],[8.999999E+09,8.999999E+09,8.999999E+09,8.999999E+09,8.999999E+09,8.999999E+09]];
    LOCAL CONST Robtarget Tr_meulage_motif_2_58 := [[-43.76195703125,-137.739,5.16978271484375],[-0.000274293000079729,0.00605508420207388,-0.0452523792521339,-0.998957197727048],[0,0,0,0],[8.999999E+09,8.999999E+09,8.999999E+09,8.999999E+09,8.999999E+09,8.999999E+09]];
    LOCAL CONST Robtarget Tr_meulage_motif_2_59 := [[-43.84648046875,-136.564140625,5.04001806640625],[-0.000274293000079729,0.00605508420207388,-0.0452523792521339,-0.998957197727048],[0,0,0,0],[8.999999E+09,8.999999E+09,8.999999E+09,8.999999E+09,8.999999E+09,8.999999E+09]];
    LOCAL CONST Robtarget Tr_meulage_motif_2_60 := [[-44.075640625,-135.88834375,4.966064453125],[-0.000274293000079729,0.00605508420207388,-0.0452523792521339,-0.998957197727048],[0,0,0,0],[8.999999E+09,8.999999E+09,8.999999E+09,8.999999E+09,8.999999E+09,8.999999E+09]];
    LOCAL CONST Robtarget Tr_meulage_motif_2_61 := [[-44.6714453125,-134.79071875,4.8468017578125],[-0.000274293000079729,0.00605508420207388,-0.0452523792521339,-0.998957197727048],[0,0,0,0],[8.999999E+09,8.999999E+09,8.999999E+09,8.999999E+09,8.999999E+09,8.999999E+09]];
    LOCAL CONST Robtarget Tr_meulage_motif_2_62 := [[-45.113890625,-134.229234375,4.786318359375],[-0.000274293000079729,0.00605508420207388,-0.0452523792521339,-0.998957197727048],[0,0,0,0],[8.999999E+09,8.999999E+09,8.999999E+09,8.999999E+09,8.999999E+09,8.999999E+09]];
    LOCAL CONST Robtarget Tr_meulage_motif_2_63 := [[-46.0290703125,-133.392421875,4.69715234375],[-0.000274293000079729,0.00605508420207388,-0.0452523792521339,-0.998957197727048],[0,0,0,0],[8.999999E+09,8.999999E+09,8.999999E+09,8.999999E+09,8.999999E+09,8.999999E+09]];
    LOCAL CONST Robtarget Tr_meulage_motif_2_64 := [[-46.73540234375,-132.87565625,4.64262744140625],[-0.000274293000079729,0.00605508420207388,-0.0452523792521339,-0.998957197727048],[0,0,0,0],[8.999999E+09,8.999999E+09,8.999999E+09,8.999999E+09,8.999999E+09,8.999999E+09]];
    LOCAL CONST Robtarget Tr_meulage_motif_2_65 := [[-47.56976171875,-132.41521875,4.594828125],[-0.000274293000079729,0.00605508420207388,-0.0452523792521339,-0.998957197727048],[0,0,0,0],[8.999999E+09,8.999999E+09,8.999999E+09,8.999999E+09,8.999999E+09,8.999999E+09]];
    LOCAL CONST Robtarget Tr_meulage_motif_2_66 := [[-48.47906640625,-132.031953125,4.555857421875],[-0.000274293000079729,0.00605508420207388,-0.0452523792521339,-0.998957197727048],[0,0,0,0],[8.999999E+09,8.999999E+09,8.999999E+09,8.999999E+09,8.999999E+09,8.999999E+09]];
    LOCAL CONST Robtarget Tr_meulage_motif_2_67 := [[-49.39833984375,-131.643640625,4.5163671875],[-0.000274293000079729,0.00605508420207388,-0.0452523792521339,-0.998957197727048],[0,0,0,0],[8.999999E+09,8.999999E+09,8.999999E+09,8.999999E+09,8.999999E+09,8.999999E+09]];
    LOCAL CONST Robtarget Tr_meulage_motif_2_68 := [[-50.356421875,-131.3585,4.48844921875],[-0.000274293000079729,0.00605508420207388,-0.0452523792521339,-0.998957197727048],[0,0,0,0],[8.999999E+09,8.999999E+09,8.999999E+09,8.999999E+09,8.999999E+09,8.999999E+09]];
    LOCAL CONST Robtarget Tr_meulage_motif_2_69 := [[-51.31450390625,-131.073375,4.46053125],[-0.000274293000079729,0.00605508420207388,-0.0452523792521339,-0.998957197727048],[0,0,0,0],[8.999999E+09,8.999999E+09,8.999999E+09,8.999999E+09,8.999999E+09,8.999999E+09]];
    LOCAL CONST Robtarget Tr_meulage_motif_2_70 := [[-52.2725859375,-130.788234375,4.43261376953125],[-0.000274293000079729,0.00605508420207388,-0.0452523792521339,-0.998957197727048],[0,0,0,0],[8.999999E+09,8.999999E+09,8.999999E+09,8.999999E+09,8.999999E+09,8.999999E+09]];
    LOCAL CONST Robtarget Tr_meulage_motif_2_71 := [[-53.23066796875,-130.5031015625,4.40469580078125],[-0.000274293000079729,0.00605508420207388,-0.0452523792521339,-0.998957197727048],[0,0,0,0],[8.999999E+09,8.999999E+09,8.999999E+09,8.999999E+09,8.999999E+09,8.999999E+09]];
    LOCAL CONST Robtarget Tr_meulage_motif_2_72 := [[-54.18874609375,-130.21796875,4.37677783203125],[-0.000274293000079729,0.00605508420207388,-0.0452523792521339,-0.998957197727048],[0,0,0,0],[8.999999E+09,8.999999E+09,8.999999E+09,8.999999E+09,8.999999E+09,8.999999E+09]];
    LOCAL CONST Robtarget Tr_meulage_motif_2_73 := [[-55.146828125,-129.9328359375,4.3488603515625],[-0.000274293000079729,0.00605508420207388,-0.0452523792521339,-0.998957197727048],[0,0,0,0],[8.999999E+09,8.999999E+09,8.999999E+09,8.999999E+09,8.999999E+09,8.999999E+09]];
    LOCAL CONST Robtarget Tr_meulage_motif_2_74 := [[-56.10491015625,-129.647703125,4.3209423828125],[-0.000274293000079729,0.00605508420207388,-0.0452523792521339,-0.998957197727048],[0,0,0,0],[8.999999E+09,8.999999E+09,8.999999E+09,8.999999E+09,8.999999E+09,8.999999E+09]];
    LOCAL CONST Robtarget Tr_meulage_motif_2_75 := [[-57.0629921875,-129.3625703125,4.29302490234375],[-0.000274293000079729,0.00605508420207388,-0.0452523792521339,-0.998957197727048],[0,0,0,0],[8.999999E+09,8.999999E+09,8.999999E+09,8.999999E+09,8.999999E+09,8.999999E+09]];
    LOCAL CONST Robtarget Tr_meulage_motif_2_76 := [[-58.02107421875,-129.0774375,4.26510693359375],[-0.000274293000079729,0.00605508420207388,-0.0452523792521339,-0.998957197727048],[0,0,0,0],[8.999999E+09,8.999999E+09,8.999999E+09,8.999999E+09,8.999999E+09,8.999999E+09]];
    LOCAL CONST Robtarget Tr_meulage_motif_2_77 := [[-58.97915234375,-128.7923046875,4.23718896484375],[-0.000274293000079729,0.00605508420207388,-0.0452523792521339,-0.998957197727048],[0,0,0,0],[8.999999E+09,8.999999E+09,8.999999E+09,8.999999E+09,8.999999E+09,8.999999E+09]];
    LOCAL CONST Robtarget Tr_meulage_motif_2_78 := [[-59.89842578125,-128.4039921875,4.19769873046875],[-0.000274293000079729,0.00605508420207388,-0.0452523792521339,-0.998957197727048],[0,0,0,0],[8.999999E+09,8.999999E+09,8.999999E+09,8.999999E+09,8.999999E+09,8.999999E+09]];
    LOCAL CONST Robtarget Tr_meulage_motif_2_79 := [[-60.74475390625,-127.93303125,4.14877880859375],[-0.000274293000079729,0.00605508420207388,-0.0452523792521339,-0.998957197727048],[0,0,0,0],[8.999999E+09,8.999999E+09,8.999999E+09,8.999999E+09,8.999999E+09,8.999999E+09]];
    LOCAL CONST Robtarget Tr_meulage_motif_2_80 := [[-61.4838515625,-127.4310546875,4.09601611328125],[-0.000274293000079729,0.00605508420207388,-0.0452523792521339,-0.998957197727048],[0,0,0,0],[8.999999E+09,8.999999E+09,8.999999E+09,8.999999E+09,8.999999E+09,8.999999E+09]];
    LOCAL CONST Robtarget Tr_meulage_motif_2_81 := [[-62.1233046875,-126.9544921875,4.04568701171875],[-0.000274293000079729,0.00605508420207388,-0.0452523792521339,-0.998957197727048],[0,0,0,0],[8.999999E+09,8.999999E+09,8.999999E+09,8.999999E+09,8.999999E+09,8.999999E+09]];
    LOCAL CONST Robtarget Tr_meulage_motif_2_82 := [[-63.00170703125,-126.0538984375,3.949318359375],[-0.000274293000079729,0.00605508420207388,-0.0452523792521339,-0.998957197727048],[0,0,0,0],[8.999999E+09,8.999999E+09,8.999999E+09,8.999999E+09,8.999999E+09,8.999999E+09]];
    LOCAL CONST Robtarget Tr_meulage_motif_2_83 := [[-63.6622265625,-124.9299140625,3.8273837890625],[-0.000274293000079729,0.00605508420207388,-0.0452523792521339,-0.998957197727048],[0,0,0,0],[8.999999E+09,8.999999E+09,8.999999E+09,8.999999E+09,8.999999E+09,8.999999E+09]];
    LOCAL CONST Robtarget Tr_meulage_motif_2_84 := [[-63.9347109375,-123.722203125,3.6946982421875],[-0.000274293000079729,0.00605508420207388,-0.0452523792521339,-0.998957197727048],[0,0,0,0],[8.999999E+09,8.999999E+09,8.999999E+09,8.999999E+09,8.999999E+09,8.999999E+09]];
    LOCAL CONST Robtarget Tr_meulage_motif_2_85 := [[-63.8149296875,-122.7366484375,3.58511645507813],[-0.000274293000079729,0.00605508420207388,-0.0452523792521339,-0.998957197727048],[0,0,0,0],[8.999999E+09,8.999999E+09,8.999999E+09,8.999999E+09,8.999999E+09,8.999999E+09]];
    LOCAL CONST Robtarget Tr_meulage_motif_2_86 := [[-63.63034375,-122.5792734375,3.56698681640625],[-0.000274293000079729,0.00605508420207388,-0.0452523792521339,-0.998957197727048],[0,0,0,0],[8.999999E+09,8.999999E+09,8.999999E+09,8.999999E+09,8.999999E+09,8.999999E+09]];
    LOCAL CONST Robtarget Tr_meulage_motif_2_87 := [[-63.304046875,-121.9228046875,3.49305493164062],[-0.000274293000079729,0.00605508420207388,-0.0452523792521339,-0.998957197727048],[0,0,0,0],[8.999999E+09,8.999999E+09,8.999999E+09,8.999999E+09,8.999999E+09,8.999999E+09]];
    LOCAL CONST Robtarget Tr_meulage_motif_2_88 := [[-62.3803203125,-121.225765625,3.41235205078125],[-0.000274293000079729,0.00605508420207388,-0.0452523792521339,-0.998957197727048],[0,0,0,0],[8.999999E+09,8.999999E+09,8.999999E+09,8.999999E+09,8.999999E+09,8.999999E+09]];
    LOCAL CONST Robtarget Tr_meulage_motif_2_89 := [[-61.713203125,-120.943140625,3.3785146484375],[-0.000274293000079729,0.00605508420207388,-0.0452523792521339,-0.998957197727048],[0,0,0,0],[8.999999E+09,8.999999E+09,8.999999E+09,8.999999E+09,8.999999E+09,8.999999E+09]];
    LOCAL CONST Robtarget Tr_meulage_motif_2_90 := [[-60.47831640625,-120.760375,3.35356860351563],[-0.000274293000079729,0.00605508420207388,-0.0452523792521339,-0.998957197727048],[0,0,0,0],[8.999999E+09,8.999999E+09,8.999999E+09,8.999999E+09,8.999999E+09,8.999999E+09]];
    LOCAL CONST Robtarget Tr_meulage_motif_2_91 := [[-59.59305078125,-120.7498671875,3.34902880859375],[-0.000274293000079729,0.00605508420207388,-0.0452523792521339,-0.998957197727048],[0,0,0,0],[8.999999E+09,8.999999E+09,8.999999E+09,8.999999E+09,8.999999E+09,8.999999E+09]];
    LOCAL CONST Robtarget Tr_meulage_motif_2_92 := [[-58.64154296875,-120.820921875,3.35326831054688],[-0.000274293000079729,0.00605508420207388,-0.0452523792521339,-0.998957197727048],[0,0,0,0],[8.999999E+09,8.999999E+09,8.999999E+09,8.999999E+09,8.999999E+09,8.999999E+09]];
    LOCAL CONST Robtarget Tr_meulage_motif_2_93 := [[-57.67001953125,-120.99740625,3.36910400390625],[-0.000274293000079729,0.00605508420207388,-0.0452523792521339,-0.998957197727048],[0,0,0,0],[8.999999E+09,8.999999E+09,8.999999E+09,8.999999E+09,8.999999E+09,8.999999E+09]];
    LOCAL CONST Robtarget Tr_meulage_motif_2_94 := [[-56.6873828125,-121.1751171875,3.38503369140625],[-0.000274293000079729,0.00605508420207388,-0.0452523792521339,-0.998957197727048],[0,0,0,0],[8.999999E+09,8.999999E+09,8.999999E+09,8.999999E+09,8.999999E+09,8.999999E+09]];
    LOCAL CONST Robtarget Tr_meulage_motif_2_95 := [[-55.72930078125,-121.46025,3.41295141601563],[-0.000274293000079729,0.00605508420207388,-0.0452523792521339,-0.998957197727048],[0,0,0,0],[8.999999E+09,8.999999E+09,8.999999E+09,8.999999E+09,8.999999E+09,8.999999E+09]];
    LOCAL CONST Robtarget Tr_meulage_motif_2_96 := [[-54.77121875,-121.7453828125,3.44086938476562],[-0.000274293000079729,0.00605508420207388,-0.0452523792521339,-0.998957197727048],[0,0,0,0],[8.999999E+09,8.999999E+09,8.999999E+09,8.999999E+09,8.999999E+09,8.999999E+09]];
    LOCAL CONST Robtarget Tr_meulage_motif_2_97 := [[-53.81313671875,-122.030515625,3.468787109375],[-0.000274293000079729,0.00605508420207388,-0.0452523792521339,-0.998957197727048],[0,0,0,0],[8.999999E+09,8.999999E+09,8.999999E+09,8.999999E+09,8.999999E+09,8.999999E+09]];
    LOCAL CONST Robtarget Tr_meulage_motif_2_98 := [[-52.8550546875,-122.3156484375,3.49670483398438],[-0.000274293000079729,0.00605508420207388,-0.0452523792521339,-0.998957197727048],[0,0,0,0],[8.999999E+09,8.999999E+09,8.999999E+09,8.999999E+09,8.999999E+09,8.999999E+09]];
    LOCAL CONST Robtarget Tr_meulage_motif_2_99 := [[-51.8969765625,-122.60078125,3.52462255859375],[-0.000274293000079729,0.00605508420207388,-0.0452523792521339,-0.998957197727048],[0,0,0,0],[8.999999E+09,8.999999E+09,8.999999E+09,8.999999E+09,8.999999E+09,8.999999E+09]];
    LOCAL CONST Robtarget Tr_meulage_motif_2_100 := [[-50.93889453125,-122.8859140625,3.55254052734375],[-0.000274293000079729,0.00605508420207388,-0.0452523792521339,-0.998957197727048],[0,0,0,0],[8.999999E+09,8.999999E+09,8.999999E+09,8.999999E+09,8.999999E+09,8.999999E+09]];
    LOCAL CONST Robtarget Tr_meulage_motif_2_101 := [[-49.9808125,-123.171046875,3.58045825195313],[-0.000274293000079729,0.00605508420207388,-0.0452523792521339,-0.998957197727048],[0,0,0,0],[8.999999E+09,8.999999E+09,8.999999E+09,8.999999E+09,8.999999E+09,8.999999E+09]];
    LOCAL CONST Robtarget Tr_meulage_motif_2_102 := [[-49.02273046875,-123.4561796875,3.6083759765625],[-0.000274293000079729,0.00605508420207388,-0.0452523792521339,-0.998957197727048],[0,0,0,0],[8.999999E+09,8.999999E+09,8.999999E+09,8.999999E+09,8.999999E+09,8.999999E+09]];
    LOCAL CONST Robtarget Tr_meulage_motif_2_103 := [[-48.0646484375,-123.7413125,3.63629370117188],[-0.000274293000079729,0.00605508420207388,-0.0452523792521339,-0.998957197727048],[0,0,0,0],[8.999999E+09,8.999999E+09,8.999999E+09,8.999999E+09,8.999999E+09,8.999999E+09]];
    LOCAL CONST Robtarget Tr_meulage_motif_2_104 := [[-47.1065703125,-124.0264453125,3.66421166992188],[-0.000274293000079729,0.00605508420207388,-0.0452523792521339,-0.998957197727048],[0,0,0,0],[8.999999E+09,8.999999E+09,8.999999E+09,8.999999E+09,8.999999E+09,8.999999E+09]];
    LOCAL CONST Robtarget Tr_meulage_motif_2_105 := [[-46.14848828125,-124.311578125,3.69212939453125],[-0.000274293000079729,0.00605508420207388,-0.0452523792521339,-0.998957197727048],[0,0,0,0],[8.999999E+09,8.999999E+09,8.999999E+09,8.999999E+09,8.999999E+09,8.999999E+09]];
    LOCAL CONST Robtarget Tr_meulage_motif_2_106 := [[-45.19040625,-124.5967109375,3.72004711914063],[-0.000274293000079729,0.00605508420207388,-0.0452523792521339,-0.998957197727048],[0,0,0,0],[8.999999E+09,8.999999E+09,8.999999E+09,8.999999E+09,8.999999E+09,8.999999E+09]];
    LOCAL CONST Robtarget Tr_meulage_motif_2_107 := [[-44.23232421875,-124.88184375,3.74796484375],[-0.000274293000079729,0.00605508420207388,-0.0452523792521339,-0.998957197727048],[0,0,0,0],[8.999999E+09,8.999999E+09,8.999999E+09,8.999999E+09,8.999999E+09,8.999999E+09]];
    LOCAL CONST Robtarget Tr_meulage_motif_2_108 := [[-43.2742421875,-125.1669765625,3.7758828125],[-0.000274293000079729,0.00605508420207388,-0.0452523792521339,-0.998957197727048],[0,0,0,0],[8.999999E+09,8.999999E+09,8.999999E+09,8.999999E+09,8.999999E+09,8.999999E+09]];
    LOCAL CONST Robtarget Tr_meulage_motif_2_109 := [[-42.3161640625,-125.452109375,3.80380053710938],[-0.000274293000079729,0.00605508420207388,-0.0452523792521339,-0.998957197727048],[0,0,0,0],[8.999999E+09,8.999999E+09,8.999999E+09,8.999999E+09,8.999999E+09,8.999999E+09]];
    LOCAL CONST Robtarget Tr_meulage_motif_2_110 := [[-41.35808203125,-125.7372421875,3.83171826171875],[-0.000274293000079729,0.00605508420207388,-0.0452523792521339,-0.998957197727048],[0,0,0,0],[8.999999E+09,8.999999E+09,8.999999E+09,8.999999E+09,8.999999E+09,8.999999E+09]];
    LOCAL CONST Robtarget Tr_meulage_motif_2_111 := [[-40.4,-126.022375,3.85963598632812],[-0.000274293000079729,0.00605508420207388,-0.0452523792521339,-0.998957197727048],[0,0,0,0],[8.999999E+09,8.999999E+09,8.999999E+09,8.999999E+09,8.999999E+09,8.999999E+09]];
    LOCAL CONST Robtarget Tr_meulage_motif_2_112 := [[-39.44191796875,-126.3075078125,3.88755395507813],[-0.000274293000079729,0.00605508420207388,-0.0452523792521339,-0.998957197727048],[0,0,0,0],[8.999999E+09,8.999999E+09,8.999999E+09,8.999999E+09,8.999999E+09,8.999999E+09]];
    LOCAL CONST Robtarget Tr_meulage_motif_2_113 := [[-38.4838359375,-126.592640625,3.9154716796875],[-0.000274293000079729,0.00605508420207388,-0.0452523792521339,-0.998957197727048],[0,0,0,0],[8.999999E+09,8.999999E+09,8.999999E+09,8.999999E+09,8.999999E+09,8.999999E+09]];
    LOCAL CONST Robtarget Tr_meulage_motif_2_114 := [[-37.5257578125,-126.8777734375,3.94338940429687],[-0.000274293000079729,0.00605508420207388,-0.0452523792521339,-0.998957197727048],[0,0,0,0],[8.999999E+09,8.999999E+09,8.999999E+09,8.999999E+09,8.999999E+09,8.999999E+09]];
    LOCAL CONST Robtarget Tr_meulage_motif_2_115 := [[-36.56767578125,-127.16290625,3.97130737304688],[-0.000274293000079729,0.00605508420207388,-0.0452523792521339,-0.998957197727048],[0,0,0,0],[8.999999E+09,8.999999E+09,8.999999E+09,8.999999E+09,8.999999E+09,8.999999E+09]];

